// TIA Portal project "FactoryIO_Template_S7-1200_V15_V16" (V16)
// Vorlageprojekt für das Buch mit Zielsystem S7-1200

(* hardware
DEVICE "S7-1200-Station_1"  S7-1200 Station
   slot 0: "Baugruppenträger_0"  Rack  V1.0
   slot 1: "PLC_1"  CPU 1211C DC/DC/DC  6ES7 211-1AE40-0XB0  V4.1
*)

// ===== PLC "PLC_1"  CPU 1211C DC/DC/DC =====

VAR_GLOBAL   // PLC tag table "Standard-Variablentabelle"
   "Tag_1" AT %A0.0 : Bool;
   "Tag_2" AT %E0.0 : Bool;
   "Tag_3" AT %E0.1 : Bool;
   "System_Byte" AT %MB1 : Byte;
   "FirstScan" AT %M1.0 : Bool;
   "DiagStatusUpdate" AT %M1.1 : Bool;
   "AlwaysTRUE" AT %M1.2 : Bool;
   "AlwaysFALSE" AT %M1.3 : Bool;
   "Clock_Byte" AT %MB0 : Byte;
   "Clock_10Hz" AT %M0.0 : Bool;
   "Clock_5Hz" AT %M0.1 : Bool;
   "Clock_2.5Hz" AT %M0.2 : Bool;
   "Clock_2Hz" AT %M0.3 : Bool;
   "Clock_1.25Hz" AT %M0.4 : Bool;
   "Clock_1Hz" AT %M0.5 : Bool;
   "Clock_0.625Hz" AT %M0.6 : Bool;
   "Clock_0.5Hz" AT %M0.7 : Bool;
END_VAR

VAR_GLOBAL   // PLC tag table "factory io"
   "伸出收料到位" AT %I0.2 : Bool;
   "叉车在中间" AT %I0.3 : Bool;
   "伸出放料到位" AT %I0.4 : Bool;
   "物料到位检测信号" AT %I0.5 : Bool;
   "检测物料开关" AT %I0.6 : Bool;
   "MovingX" AT %I0.7 : Bool;
   "Moving Z" AT %I1.0 : Bool;
   "启动" AT %I1.1 : Bool;
   "停止" AT %I1.2 : Bool;
   "出料检测传感器" AT %I1.3 : Bool;
   "显示屏传感器" AT %I1.4 : Bool;
   "复位" AT %I1.5 : Bool;
   "急停" AT %I1.6 : Bool;
   "手动模式" AT %I1.7 : Bool;
   "自动模式" AT %I2.0 : Bool;
   "FACTORY I/O (Running)" AT %I2.1 : Bool;
   "一段电机" AT %Q0.2 : Bool;
   "二段电机" AT %Q0.3 : Bool;
   "伸出取料" AT %Q0.4 : Bool;
   "叉车上升" AT %Q0.5 : Bool;
   "发料" AT %Q0.6 : Bool;
   "伸出放料" AT %Q0.7 : Bool;
   "绿色" AT %Q1.0 : Bool;
   "红色" AT %Q1.1 : Bool;
   "三段电机" AT %Q1.2 : Bool;
   "四段电机" AT %Q1.3 : Bool;
   "出料" AT %Q1.4 : Bool;
   "移动目标" AT %QD30 : DInt;
END_VAR

DATA_BLOCK "块_自动入库_DB_1"   // DB3
{ S7_Optimized_Access := 'TRUE' }
VERSION : 0.1
// stored: InstanceOfName 块_自动入库
"块_自动入库"
BEGIN
END_DATA_BLOCK

// folder: 数据块

DATA_BLOCK "数据块_自动入库"   // DB1
{ S7_Optimized_Access := 'TRUE' }
VERSION : 0.1
   VAR
      自动入库 : Struct
         置位复位优先指令 : Array[1..10] of Bool;
         定时器 : Array[1..10] of IEC_TIMER;
         放料数目 : DInt;
         沿时指令 : Array[1..10] of Bool;
         完成标志位 : Bool;
      END_STRUCT;
   END_VAR
BEGIN
   // 自动入库.置位复位优先指令[1] : 1
   // 自动入库.定时器[1] : 1
   // 自动入库.定时器[2] : 1
   // 自动入库.置位复位优先指令[2] : 1
   // 自动入库.定时器[3] : 1
   // 自动入库.置位复位优先指令[3] : 1
   // 自动入库.定时器[4] : 1
   // 自动入库.沿时指令[1] : 1
   // 自动入库.沿时指令[2] : 1
   // 自动入库.定时器[5] : 1
   // 自动入库.定时器[6] : 1
   // 自动入库.置位复位优先指令[4] : 1
   // 自动入库.沿时指令[3] : 1
END_DATA_BLOCK

// folder: (top level)

FUNCTION "MHJ-PLC-Lab-Function-S71200" : Void   // FC9000, SCL
{ S7_Optimized_Access := 'TRUE' }
VERSION : 0.1
   VAR_TEMP
      rdTimeReturn : Int;
      outputTime : DTL;
      SyncVal : Byte;
      forVal : Int;
      forVal_2 : Int;
      Value : Byte;
   END_VAR
   VAR CONSTANT
      CompVal : Byte := 16#34;
      Value_01 : Byte := 16#11;
      Value_01_DW : DWord := 16#A165_D992;
      Value_02_DW : DWord := 16#58BE_4401;
   END_VAR
BEGIN

   #Value:=PEEK(area := 16#82,
        dbNumber := 0,
        byteOffset := 511);
   #Value := #Value + 1;

   POKE(area := 16#82,
        dbNumber := 0,
        byteOffset := 511,
        value := #Value);

   POKE(area:=16#81,
        dbNumber:=0,
        byteOffset:=1016,
        value:=#Value_01_DW);
   POKE(area := 16#81,
        dbNumber := 0,
        byteOffset := 1020,
        value := #Value_02_DW);

   POKE(area := 16#81,
        dbNumber := 0,
        byteOffset := 511,
        value := B#16#00);

   FOR #forVal := 0 TO 120 DO
       FOR #forVal_2:=0 TO 10 DO
           #rdTimeReturn:=RD_SYS_T(#outputTime);
           #rdTimeReturn := WR_SYS_T(#outputTime);
           #rdTimeReturn := RD_SYS_T(#outputTime);
           #rdTimeReturn := WR_SYS_T(#outputTime);
       END_FOR;
       #SyncVal:= PEEK(area := 16#81,
                      dbNumber := 0,
                      byteOffset := 511);
       IF #SyncVal = #CompVal THEN
          GOTO M_1;
       END_IF;
   END_FOR;
   RETURN;

   M_1:
   POKE(area := 16#81,
        dbNumber := 0,
        byteOffset := 511,
        value := B#16#0);
END_FUNCTION

ORGANIZATION_BLOCK "Main"   // OB1, LAD, ProgramCycle
TITLE = "Main Program Sweep (Cycle)"
{ S7_Optimized_Access := 'TRUE' }
VERSION : 0.1
   VAR_INPUT
      Initial_Call : Bool;   // Initial call of this OB
      Remanence : Bool;   // =True, if remanent data are available
   END_VAR
BEGIN

REGION Network 1: Konnektierungsbaustein für PLC-Lab
   // Im Netzwerk 1 wird der Konnektierungsbaustein für PLC-Lab aufgerufen.
   // Dieser Aufruf darf nicht entfernt werden!
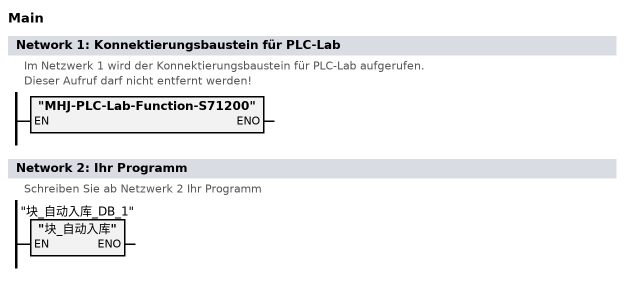
   RUNG wire#powerrail
      "MHJ-PLC-Lab-Function-S71200"()
   END_RUNG
   // the same network as SCL:
   "MHJ-PLC-Lab-Function-S71200"();
END_REGION

REGION Network 2: Ihr Programm
   // Schreiben Sie ab Netzwerk 2 Ihr Programm
   RUNG wire#powerrail
      "块_自动入库_DB_1"()
   END_RUNG
   // the same network as SCL:
   "块_自动入库_DB_1"();   // "块_自动入库"
END_REGION
END_ORGANIZATION_BLOCK

// folder: 自动入库

FUNCTION_BLOCK "块_自动入库"   // FB1, LAD
{ S7_Optimized_Access := 'TRUE' }
VERSION : 0.1
   VAR_TEMP   // added for the SCL form of the ladder/FBD networks
      _w1 : Bool;
      _w2 : Bool;
      _w3 : Bool;
   END_VAR
BEGIN

REGION Network 1: 初始化
   // 启动执行程序时，第一次执行程序，M1.0为自动置为1，来达到清零的效果，也要将升降机的数目清0
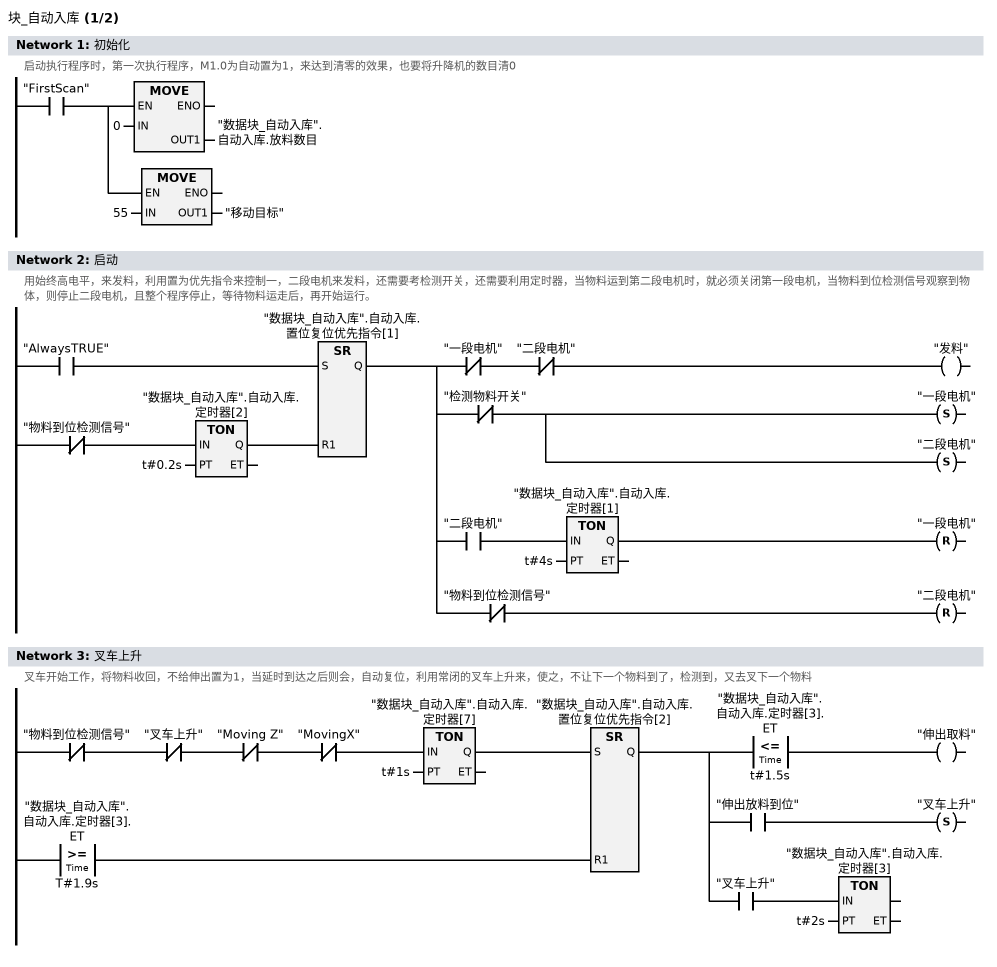
   RUNG wire#powerrail
      Contact( "FirstScan" )
      wire#w1
      Move(in := 0, out1 => "数据块_自动入库".自动入库.放料数目)
   END_RUNG
   RUNG wire#w1
      Move(in := 55, out1 => "移动目标")
   END_RUNG
   // the same network as SCL:
   IF "FirstScan" THEN
       "数据块_自动入库".自动入库.放料数目 := 0;
       "移动目标" := 55;
   END_IF;
END_REGION

REGION Network 2: 启动
   // 用始终高电平，来发料，利用置为优先指令来控制一，二段电机来发料，还需要考检测开关，还需要利用定时器，当物料运到第二段电机时，就必须关闭第一段电机，当物料到位检测信号观察到物体，则停止二段电机，且整个程序停止，等待物料运走后，再开始运行。
   "数据块_自动入库".自动入库.定时器[2].TON(IN := NOT "物料到位检测信号", PT := t#0.2s);
   IF "AlwaysTRUE" THEN
       "数据块_自动入库".自动入库.置位复位优先指令[1] := TRUE;   // SR flip-flop
   END_IF;
   IF "数据块_自动入库".自动入库.定时器[2].Q THEN "数据块_自动入库".自动入库.置位复位优先指令[1] := FALSE; END_IF;
   "发料" := "数据块_自动入库".自动入库.置位复位优先指令[1] AND NOT "一段电机" AND NOT "二段电机";
   IF "数据块_自动入库".自动入库.置位复位优先指令[1] AND NOT "检测物料开关" THEN
       "一段电机" := TRUE;
       "二段电机" := TRUE;
   END_IF;
   "数据块_自动入库".自动入库.定时器[1].TON(IN := "数据块_自动入库".自动入库.置位复位优先指令[1] AND "二段电机", PT := t#4s);
   IF "数据块_自动入库".自动入库.定时器[1].Q THEN "一段电机" := FALSE; END_IF;
   IF "数据块_自动入库".自动入库.置位复位优先指令[1] AND NOT "物料到位检测信号" THEN "二段电机" := FALSE; END_IF;
END_REGION

REGION Network 3: 叉车上升
   // 叉车开始工作，将物料收回，不给伸出置为1，当延时到达之后则会，自动复位，利用常闭的叉车上升来，使之，不让下一个物料到了，检测到，又去叉下一个物料
   "数据块_自动入库".自动入库.定时器[7].TON(IN := NOT "物料到位检测信号" AND NOT "叉车上升" AND NOT "Moving Z" AND NOT "MovingX",
                           PT := t#1s);
   IF "数据块_自动入库".自动入库.定时器[7].Q THEN
       "数据块_自动入库".自动入库.置位复位优先指令[2] := TRUE;   // SR flip-flop
   END_IF;
   IF "数据块_自动入库".自动入库.定时器[3].ET >= T#1.9s THEN "数据块_自动入库".自动入库.置位复位优先指令[2] := FALSE; END_IF;
   "伸出取料" := "数据块_自动入库".自动入库.置位复位优先指令[2] AND ("数据块_自动入库".自动入库.定时器[3].ET <= t#1.5s);
   IF "数据块_自动入库".自动入库.置位复位优先指令[2] AND "伸出放料到位" THEN "叉车上升" := TRUE; END_IF;
   "数据块_自动入库".自动入库.定时器[3].TON(IN := "数据块_自动入库".自动入库.置位复位优先指令[2] AND "叉车上升", PT := t#2s);
END_REGION

REGION Network 4: 将物料取到
   // 从最开始放物料，放料的时间会越来越长，当上面的取料置为指令复位后，通过用沿时指令来确保递增，当然沿时指令只能确保一个周期
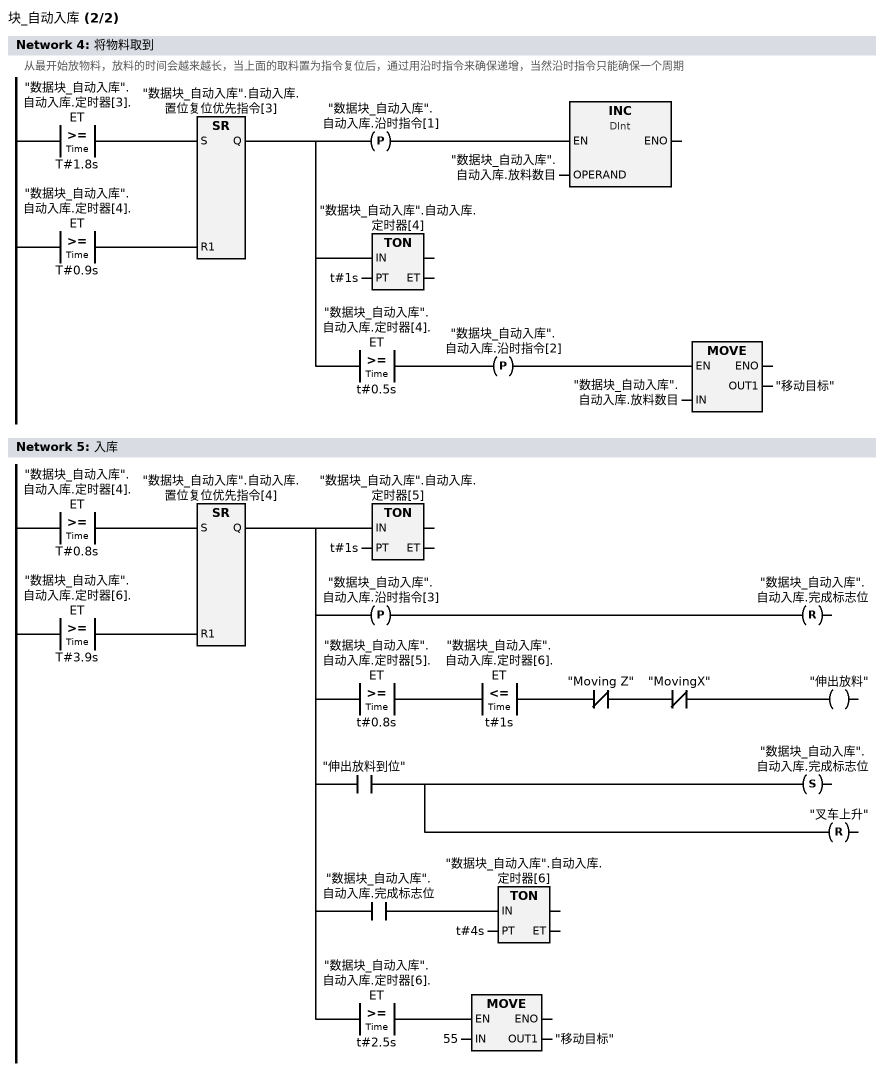
   IF "数据块_自动入库".自动入库.定时器[3].ET >= T#1.8s THEN
       "数据块_自动入库".自动入库.置位复位优先指令[3] := TRUE;   // SR flip-flop
   END_IF;
   IF "数据块_自动入库".自动入库.定时器[4].ET >= T#0.9s THEN "数据块_自动入库".自动入库.置位复位优先指令[3] := FALSE; END_IF;
   #_w1 := "数据块_自动入库".自动入库.置位复位优先指令[3] AND NOT "数据块_自动入库".自动入库.沿时指令[1];   // rising edge
   "数据块_自动入库".自动入库.沿时指令[1] := "数据块_自动入库".自动入库.置位复位优先指令[3];
   IF #_w1 THEN "数据块_自动入库".自动入库.放料数目 := "数据块_自动入库".自动入库.放料数目 + 1; END_IF;
   "数据块_自动入库".自动入库.定时器[4].TON(IN := "数据块_自动入库".自动入库.置位复位优先指令[3], PT := t#1s);
   #_w2 := "数据块_自动入库".自动入库.置位复位优先指令[3] AND ("数据块_自动入库".自动入库.定时器[4].ET >= t#0.5s);
   #_w3 := #_w2 AND NOT "数据块_自动入库".自动入库.沿时指令[2];   // rising edge
   "数据块_自动入库".自动入库.沿时指令[2] := #_w2;
   IF #_w3 THEN "移动目标" := "数据块_自动入库".自动入库.放料数目; END_IF;
END_REGION

REGION Network 5: 入库
   IF "数据块_自动入库".自动入库.定时器[4].ET >= T#0.8s THEN
       "数据块_自动入库".自动入库.置位复位优先指令[4] := TRUE;   // SR flip-flop
   END_IF;
   IF "数据块_自动入库".自动入库.定时器[6].ET >= T#3.9s THEN "数据块_自动入库".自动入库.置位复位优先指令[4] := FALSE; END_IF;
   "数据块_自动入库".自动入库.定时器[5].TON(IN := "数据块_自动入库".自动入库.置位复位优先指令[4], PT := t#1s);
   #_w1 := "数据块_自动入库".自动入库.置位复位优先指令[4] AND NOT "数据块_自动入库".自动入库.沿时指令[3];   // rising edge
   "数据块_自动入库".自动入库.沿时指令[3] := "数据块_自动入库".自动入库.置位复位优先指令[4];
   IF #_w1 THEN "数据块_自动入库".自动入库.完成标志位 := FALSE; END_IF;
   "伸出放料" := "数据块_自动入库".自动入库.置位复位优先指令[4] AND ("数据块_自动入库".自动入库.定时器[5].ET >= t#0.8s) AND ("数据块_自动入库".自动入库.定时器[6].ET <= t#1s) AND NOT "Moving Z" AND NOT "MovingX";
   IF "数据块_自动入库".自动入库.置位复位优先指令[4] AND "伸出放料到位" THEN
       "数据块_自动入库".自动入库.完成标志位 := TRUE;
       "叉车上升" := FALSE;
   END_IF;
   "数据块_自动入库".自动入库.定时器[6].TON(IN := "数据块_自动入库".自动入库.置位复位优先指令[4] AND "数据块_自动入库".自动入库.完成标志位, PT := t#4s);
   IF "数据块_自动入库".自动入库.置位复位优先指令[4] AND ("数据块_自动入库".自动入库.定时器[6].ET >= t#2.5s) THEN "移动目标" := 55; END_IF;
END_REGION
END_FUNCTION_BLOCK